FUNCTION_BLOCK Seq_3
VAR_INPUT
	// Basis-Inputs
	bExecute			:BOOL;				// Trigger für Ausführung von Sequenz
	iSysCommand			:eSystemCommand;	// Steuerungsvariabel von System (Resetten)
	iSysState			:eSystemState;		// Information über Zustand von System
	
	
	// Prozess-Inputs 
	Parameter_1			:sSmartGreiferProzessVariablen;
	Parameter_2			:sSmartGreiferProzessVariablen;
	Parameter_3			:sSmartGreiferProzessVariablen;
	Parameter_4			:sSmartGreiferProzessVariablen;
END_VAR
VAR_OUTPUT
	bDone				:BOOL;				// Information ob Sequenz ausgfeührt wurde
	bBusy				:BOOL;				// Information ob Sequenz im Moment ausgeführt wird
	bError				:BOOL;				// Information ob sich Sequenz in Fehlerzustand befindet
END_VAR
VAR
	// Sequenz-Zustände
	iState				:eSequenceState;
	
	// Startvariablen (FB soll nur bei einer steigenden Flanke gestartet werden)
	fTrigger			:R_TRIG;			// Erkennung einer steigenden Flanke für den Starte
	fSwitch				:SR;				// Setzen des Signals
	bSwitchResett		:BOOL;				// Resetten des Signals
	
	// Zustandsvariablen
	bStarten			:BOOL;
	bStoppen			:BOOL;
	bResetten			:BOOL;
	
	// Management-Variablen:
	bFinished			:BOOL;
	bInit				:BOOL;
	
	// Skill-Instanziierungen
	MoveGripper			:Skill_Greifer_Pos_Anfahren;
	CloseGripper		:Skill_Greifer_Schliessen;
	OpenGripper			:Skill_Greifer_Oeffnen;
	Parameter			:sSmartGreiferProzessVariablen;
END_VAR

// Aufrufen von Skills und Ablauf
Ablauf();	
Skills();

//_______________________________________________________________
// Reaktion auf Fehler
IF bError THEN
	iState := 3;
END_IF	

// Reaktion auf Input-Variablen: 
	// Starten
	fTrigger(CLK := bExecute);
	fSwitch(Set1 := fTrigger.Q);
	
	IF fSwitch.Q1 THEN
		bStarten := TRUE;
	ELSE
		bStarten := FALSE;
	END_IF
	
	// Stoppen
	IF iSysCommand = 3 THEN
		bStoppen := TRUE;	
	ELSE 
		bStoppen := FALSE;	
	END_IF
	
	// Stoppen
	IF iSysCommand = 4 THEN
		bResetten := TRUE;	
	ELSE 
		bResetten := FALSE;	
	END_IF



//_______________________________________________________________
// Zustandsmanagement
CASE iState OF 
	0:	// BEREIT
			// DO	
			fSwitch.RESET := FALSE;
				
			// TRANSITION
			IF bStarten THEN
				fSwitch.RESET := TRUE;
				iState := 1;																							// Starten des Objektes 
			END_IF
	// ________________________________________________________________________________			
	1:	// LAUFEND
			// DO
			bBusy := TRUE;	

			IF bStoppen THEN
				SFCReset := TRUE;
				bBusy := FALSE;
			END_IF	
			
			// TRANSITION
			IF bFinished THEN
				bFinished := FALSE;
				bBusy := FALSE;
				iState := 2;
			END_IF
			
			IF bInit THEN
				bInit := FALSE;
				SFCReset := FALSE;
				iState := 0;
			END_IF

	// ________________________________________________________________________________					
	2:	// ABGESCHLOSSEN
			// DO
			bDone := TRUE;			
						
			// TRANSITION
			IF bDone THEN
				bDone := FALSE;
				iState := 0;
			END_IF
	// ________________________________________________________________________________					
	3:	// FEHLER
			// DO
			bDone := FALSE;
			bBusy := FALSE;
			
			// TRANSITION
			IF bResetten THEN
				bError := FALSE;
				iState := 0;
			END_IF
			
END_CASE

ACTION Ablauf:
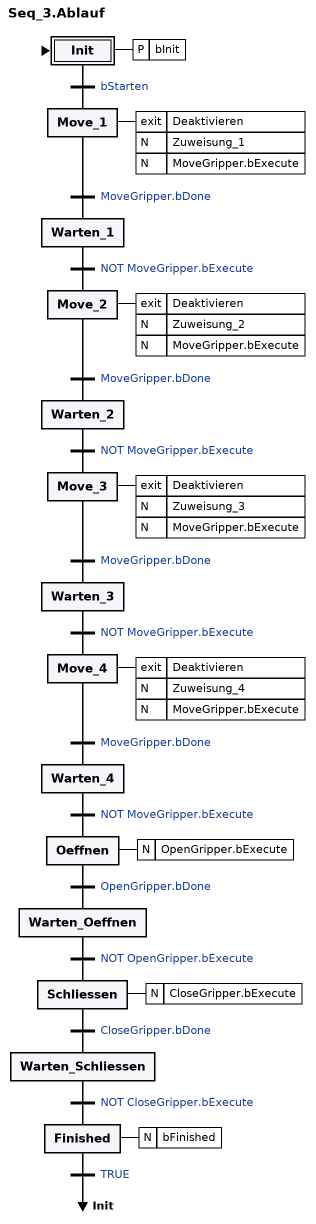
INITIAL_STEP Init:
    bInit(P);
END_STEP
TRANSITION FROM Init TO Move_1
    := bStarten;
END_TRANSITION
STEP Move_1:
    Deaktivieren(P0);  // exit action
    Zuweisung_1(N);
    MoveGripper.bExecute(N);
END_STEP
TRANSITION FROM Move_1 TO Warten_1
    := MoveGripper.bDone;
END_TRANSITION
STEP Warten_1:
END_STEP
TRANSITION FROM Warten_1 TO Move_2
    := NOT MoveGripper.bExecute;
END_TRANSITION
STEP Move_2:
    Deaktivieren(P0);  // exit action
    Zuweisung_2(N);
    MoveGripper.bExecute(N);
END_STEP
TRANSITION FROM Move_2 TO Warten_2
    := MoveGripper.bDone;
END_TRANSITION
STEP Warten_2:
END_STEP
TRANSITION FROM Warten_2 TO Move_3
    := NOT MoveGripper.bExecute;
END_TRANSITION
STEP Move_3:
    Deaktivieren(P0);  // exit action
    Zuweisung_3(N);
    MoveGripper.bExecute(N);
END_STEP
TRANSITION FROM Move_3 TO Warten_3
    := MoveGripper.bDone;
END_TRANSITION
STEP Warten_3:
END_STEP
TRANSITION FROM Warten_3 TO Move_4
    := NOT MoveGripper.bExecute;
END_TRANSITION
STEP Move_4:
    Deaktivieren(P0);  // exit action
    Zuweisung_4(N);
    MoveGripper.bExecute(N);
END_STEP
TRANSITION FROM Move_4 TO Warten_4
    := MoveGripper.bDone;
END_TRANSITION
STEP Warten_4:
END_STEP
TRANSITION FROM Warten_4 TO Oeffnen
    := NOT MoveGripper.bExecute;
END_TRANSITION
STEP Oeffnen:
    OpenGripper.bExecute(N);
END_STEP
TRANSITION FROM Oeffnen TO Warten_Oeffnen
    := OpenGripper.bDone;
END_TRANSITION
STEP Warten_Oeffnen:
END_STEP
TRANSITION FROM Warten_Oeffnen TO Schliessen
    := NOT OpenGripper.bExecute;
END_TRANSITION
STEP Schliessen:
    CloseGripper.bExecute(N);
END_STEP
TRANSITION FROM Schliessen TO Warten_Schliessen
    := CloseGripper.bDone;
END_TRANSITION
STEP Warten_Schliessen:
END_STEP
TRANSITION FROM Warten_Schliessen TO Finished
    := NOT CloseGripper.bExecute;
END_TRANSITION
STEP Finished:
    bFinished(N);
END_STEP
TRANSITION FROM Finished TO Init
    := TRUE;
END_TRANSITION
END_ACTION

ACTION Deaktivieren:
MoveGripper.bExecute := FALSE;
END_ACTION

ACTION Skills:
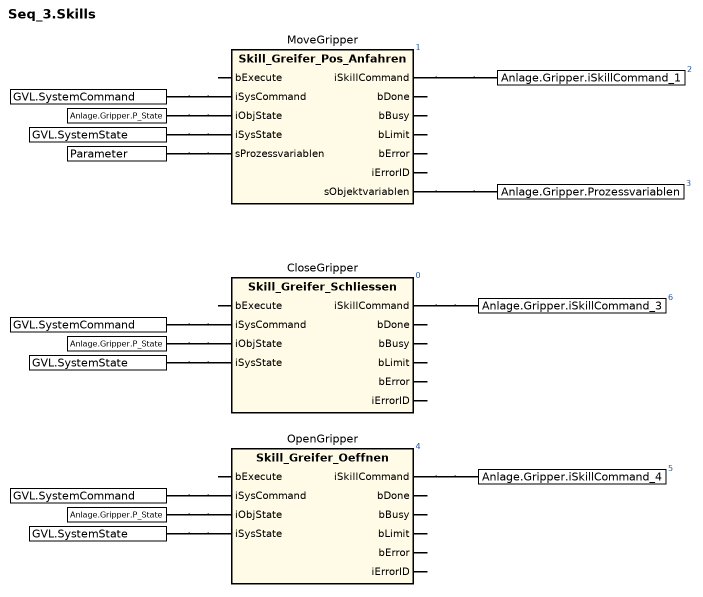
CloseGripper(
    iSysCommand := GVL.SystemCommand,
    iObjState := Anlage.Gripper.P_State,
    iSysState := GVL.SystemState); // Skill_Greifer_Schliessen
MoveGripper(
    iSysCommand := GVL.SystemCommand,
    iObjState := Anlage.Gripper.P_State,
    iSysState := GVL.SystemState,
    sProzessvariablen := Parameter); // Skill_Greifer_Pos_Anfahren
Anlage.Gripper.iSkillCommand_1 := MoveGripper.iSkillCommand;
Anlage.Gripper.Prozessvariablen := MoveGripper.sObjektvariablen;
OpenGripper(
    iSysCommand := GVL.SystemCommand,
    iObjState := Anlage.Gripper.P_State,
    iSysState := GVL.SystemState); // Skill_Greifer_Oeffnen
Anlage.Gripper.iSkillCommand_4 := OpenGripper.iSkillCommand;
Anlage.Gripper.iSkillCommand_3 := CloseGripper.iSkillCommand;
END_ACTION

ACTION Zuweisung_1:
Parameter := Parameter_1;
END_ACTION

ACTION Zuweisung_2:
Parameter := Parameter_2;
END_ACTION

ACTION Zuweisung_3:
Parameter := Parameter_3;
END_ACTION

ACTION Zuweisung_4:
Parameter := Parameter_4;
END_ACTION

END_FUNCTION_BLOCK

(* stored: Version 1.1.0.1
   POU Seq_3: Id {be2994b2-ac71-4ad5-a94a-b6ec9e2fdb31}, SpecialFunc None
   Folder 00_Hilfsaktionen: Id {212cb3a5-af12-4368-ace7-4075da4754e3}
   Folder 01_Zusweisung: Id {4be89e8f-0f35-4c80-a9fb-799a2f5f3671}
   Action Ablauf: Id {de921999-3ec1-4525-9500-59fb5e61c19e}
   Action Deaktivieren: Id {5381399d-2150-4448-b7d5-5f7962e795bd}
   Action Skills: Id {0cd82750-6c56-4654-ab52-353456f46a6a}
   Action Zuweisung_1: Id {319397ca-4a5b-43c0-8f40-967db70b2c39}
   Action Zuweisung_2: Id {ff65ad65-1135-4e82-872b-26e530cf89d8}
   Action Zuweisung_3: Id {62c7d830-0881-41d9-a92d-1d5263fedcbb}
   Action Zuweisung_4: Id {648c2b30-c536-4662-b8c0-dacf3bb1ee75} *)
